PROGRAM MAIN
VAR
	fbFeeder1		: FB_Feeder(nFeederId := 1);
	fbFeeder2		: FB_Feeder(nFeederId := 2);
	bTest AT %I* : BOOL;
END_VAR

fbFeeder1();
fbFeeder2();

END_PROGRAM

(* stored: Version 1.1.0.1, ProductVersion 3.1.4024.12
   POU MAIN: Id {4e4178e0-7104-4b3d-8342-d5a78fcb71f7}, SpecialFunc None *)
